// TwinCAT 3 PLC project MyPlcProject
// ProgramVersion: 3.1.4023.0
// libraries:
//   Tc2_Standard, * (Beckhoff Automation GmbH)
//   Tc2_System, * (Beckhoff Automation GmbH)
//   Tc3_Module, * (Beckhoff Automation GmbH)
// project tree:
//   DUTs/ ST_ExampleStruct.TcDUT
//   GVLs/ GVL_Main.TcGVL
//   / PlcTask.TcTTO
//   POUs/ExampleFolder/ FB_ExampleFolder_FunctionBlock.TcPOU, F_ExampleFolder_Function.TcPOU, ST_ExampleFolder_Struct.TcDUT
//   POUs/ FB_ExampleFunctionBlock.TcPOU, F_ExampleFunction.TcPOU, MAIN.TcPOU
// real-time tasks:
//   TASK PlcTask: cycle T#10ms, priority 20, ADS port 350

CONFIGURATION MyPlcProject
    RESOURCE PLC ON TwinCAT3
        TASK PlcTask(INTERVAL := T#10ms, PRIORITY := 20);
        PROGRAM MAIN WITH PlcTask : MAIN;
    END_RESOURCE
END_CONFIGURATION

// ---- DUTs/ST_ExampleStruct.TcDUT
(*
A definition of a struct.
*)
TYPE ST_ExampleStruct :
STRUCT
    someDouble          : LREAL;        // Use to store a number
    someBoolean         : BOOL;         // Use as a flag
END_STRUCT
END_TYPE

// ---- POUs/ExampleFolder/ST_ExampleFolder_Struct.TcDUT
(*
Struct inside ExampleFolder.
*)
TYPE ST_ExampleFolder_Struct :
STRUCT
END_STRUCT
END_TYPE

// ---- GVLs/GVL_Main.TcGVL
{attribute 'qualified_only'}
VAR_GLOBAL
    flag        : BOOL;             // Flag for the system
    counter     : ULINT;            // Main counter
    cycleTIme   : LREAL := 0.001;   // Time between PLC cycles
END_VAR

// ---- POUs/MAIN.TcPOU
PROGRAM MAIN
VAR
END_VAR

END_PROGRAM

// ---- POUs/ExampleFolder/FB_ExampleFolder_FunctionBlock.TcPOU
(*
FB indside folder `ExampleFolder`.
*)
FUNCTION_BLOCK FB_ExampleFolder_FunctionBlock

METHOD ExampleFolder_FunctionBlock_Method : BOOL
VAR_INPUT
    input           : BOOL;
END_VAR
END_METHOD

END_FUNCTION_BLOCK

// ---- POUs/ExampleFolder/F_ExampleFolder_Function.TcPOU
(*
Function indside folder `ExampleFolder`.
*)
FUNCTION F_ExampleFolder_Function : BOOL

END_FUNCTION

// ---- POUs/FB_ExampleFunctionBlock.TcPOU
(*
Here we describe a function block, including some children.
*)
FUNCTION_BLOCK FB_ExampleFunctionBlock
VAR_INPUT
    input       : BOOL;
END_VAR
VAR_OUTPUT
    output      : STRING(15);
END_VAR

(*
Child method of our FB.
*)
METHOD ExampleMethod
VAR_INPUT
END_VAR
END_METHOD

(*
Reference to a variable that might be read-only.
*)
PROPERTY ExampleProperty : REFERENCE TO LREAL
GET
END_GET
SET
END_SET
END_PROPERTY

END_FUNCTION_BLOCK

// ---- POUs/F_ExampleFunction.TcPOU
(*
This is an example function block.

Here follows a longer description. 
*)
FUNCTION F_ExampleFunction : LREAL
VAR_INPUT
    inputVar1               : UDINT;                // Description of first input
    inputVar2               : REAL := 3.14;         // Description of second input
END_VAR

F_ExampleFunction := 0.0;

END_FUNCTION
